FUNCTION_BLOCK FB_Runtime
VAR_INPUT
	gotime: BOOL;
	settime: TIME;
	countdown: BOOL; // New input
	resetToTime : TIME;
END_VAR
VAR_OUTPUT
	elapsedtime: TIME;
	elapsed: BOOL;
END_VAR
VAR
	reset: BOOL;
	_resetTOTime : TIME;
	initial : BOOL := TRUE;
	presenttime: TIME;
	lasttime: TIME;
	cycletime: TIME;

END_VAR


_resetToTime := ResetToTime; 

IF initial THEN
	elapsedtime := _resetToTime;
	initial := FALSE;
END_IF

presenttime:= TIME();
IF NOT reset THEN
(* here the test of overflow*)
	IF (lasttime > presenttime) THEN (*overflow := true*);
		lasttime:= DWORD_TO_TIME(NOT TIME_TO_DWORD(lasttime))+T#1MS;
		cycletime:= presenttime+lasttime;
	ELSE
		cycletime:= presenttime - lasttime;
	END_IF
ELSE
	elapsedtime:=_resetToTime;
	cycletime:=t#0s;
END_IF

lasttime:=presenttime;

IF gotime AND NOT countDown THEN
		elapsedtime := elapsedtime + cycletime;
ELSIF NOT gotime AND countdown THEN
	IF elapsedtime > cycletime THEN
		elapsedtime := elapsedtime - cycletime;
	ELSE
		elapsedtime := T#0S;
	END_IF
END_IF

IF settime < elapsedtime THEN
	elapsed:=TRUE;
	elapsedtime := settime;
ELSE
	elapsed:=FALSE;
END_IF

reset := FALSE;

METHOD resetValues : BOOL
reset := TRUE;
END_METHOD

END_FUNCTION_BLOCK

(* stored: Version 1.1.0.1, ProductVersion 3.1.4024.9
   POU FB_Runtime: Id {2c693863-3086-4693-805e-a6f5602c35ed}, SpecialFunc None
   Method resetValues: Id {42af8755-ea1f-418c-90bb-2c804aa4483e} *)
